{attribute 'OPC.UA.DA' := '1'}
FUNCTION_BLOCK ArduinoLight EXTENDS LightBase
VAR_INPUT
END_VAR
VAR_OUTPUT
END_VAR
VAR
	{attribute 'OPC.UA.DA' := '0'}
	_config : ArduinoLightConfig;	
	{attribute 'OPC.UA.DA' := '0'}
	_coeAccess : CoeAccess;	
	{attribute 'OPC.UA.DA' := '0'}
	_initConfigSerialCom : BOOL;	
	{attribute 'OPC.UA.DA' := '0'}
	_suffix : STRING := Const.CR_LF;
	{attribute 'OPC.UA.DA' := '0'}
	_serialCom  : SerialCom(Prefix :='', Suffix := _suffix);
	{attribute 'OPC.UA.DA' := '0'}
	_refSerialCom : REFERENCE TO SerialCom(Prefix :='', Suffix := _suffix) := _serialCom;		 
	{attribute 'OPC.UA.DA' := '0'}
	_isReceived : BOOL;
	
	{attribute 'OPC.UA.DA' := '0'}
	_deliverMessages : INT;
		
	StatusMsg : STRING(255);
	SwitchOnMsg : STRING(255);
	PowerMsg : STRING(255);
	IntensityMsg : STRING(255);	
	TemperatureMsg : STRING(255);
	LightSourcesMsg : STRING(255);
	TimeLightSourceMsg  : STRING(255);
	CustomMsg : STRING(255);
		
	{region 'Commands'}
	
	{attribute 'OPC.UA.DA' := '0'}
	_setSwitchOnCmd : BOOL;
	{attribute 'OPC.UA.DA' := '0'}
	_getSwitchOnCmd : BOOL;
	{attribute 'OPC.UA.DA' := '0'}
	_setPowerCmd : BOOL;
	{attribute 'OPC.UA.DA' := '0'}
	_getPowerCmd : BOOL;
	{attribute 'OPC.UA.DA' := '0'}
	_setIntensityCmd : BOOL;
	{attribute 'OPC.UA.DA' := '0'}
	_getIntensityCmd : BOOL;
	{attribute 'OPC.UA.DA' := '0'}
	_getTimeLightSourceCmd : BOOL;
	{attribute 'OPC.UA.DA' := '0'}
	_getLightSourcesCmd : BOOL;
	{attribute 'OPC.UA.DA' := '0'}
	_customCmd : BOOL;
	{attribute 'OPC.UA.DA' := '0'}			  		   
	_raisePropertiesCmd : BOOL;
	
	{attribute 'OPC.UA.DA' := '0'}
	_lightId : STRING; 
	{attribute 'OPC.UA.DA' := '0'}
	_switchOn : BOOL;
	{attribute 'OPC.UA.DA' := '0'}
	_setPower : LREAL;
	{attribute 'OPC.UA.DA' := '0'}
	_setIntensity : LREAL;
	{attribute 'OPC.UA.DA' := '0'}
	_cmd : STRING;	
		 
	{endregion}			
	
	{attribute 'OPC.UA.DA' := '0'}
	_initDevice : BOOL;	
	 
	{attribute 'OPC.UA.DA' := '0'}
	_lightSources : ARRAY [0..Const.PHOTOLUM_NUMBER_LIGHT_SOURCE] OF STRING(255);  
	
	{attribute 'OPC.UA.DA' := '0'}
	_itemScheduler : INT;
	{attribute 'OPC.UA.DA' := '0'}
	_itemInitScheduler : INT;
	{attribute 'OPC.UA.DA' := '0'}
	_itemExecScheduler : INT;		
	{attribute 'OPC.UA.DA' := '0'}
	_itemRaisedProperties : INT;			
	{attribute 'OPC.UA.DA' := '0'}
	_pulseGenerator : TON;	
	{attribute 'OPC.UA.DA' := '0'}
	_initPulseGenerator : TON;	
	{attribute 'OPC.UA.DA' := '0'}	
	_execPulseGenerator : TON;	
	
	{attribute 'OPC.UA.DA' := '0'}
	message : STRING;
	{attribute 'OPC.UA.DA' := '0'}
	lastMessage : STRING;	
	{attribute 'OPC.UA.DA' := '0'}
	sSubStr4 : STRING(4) := '';			
	{attribute 'OPC.UA.DA' := '0'}
	stringLength : INT;
	{attribute 'OPC.UA.DA' := '0'}
	_numberOfElements : DINT;
	{attribute 'OPC.UA.DA' := '0'}
	_indexNumberOfElements : INT;
END_VAR

IF NOT InitConfigSerialCom THEN
	ConfigureSerialCom();
ELSIF THIS^.Status = TExecutionState.Ready THEN
	SUPER^();	

	IF _refSerialCom.ErrorReceiveId = COMERROR_NOERROR THEN
		_refSerialCom(TxBuffer:= HardwareGlobalVariables.TxBufferLight, 
		 	      	  RxBuffer:= HardwareGlobalVariables.RxBufferLight);
	END_IF				  
	
	// Init device
	InitDevice();		  				 
	
	IF StateMsg <> ANY_TO_STRING(State) THEN
		StateMsg := ANY_TO_STRING(State);
	END_IF
	
	// Deliver messages
	IF _refSerialCom.IsReceived THEN	
		lastMessage := _refSerialCom.LastReceivedString;			
		stringLength := LEN(lastMessage);
		
		IF stringLength > 2 THEN
			message := LEFT(lastMessage, stringLength - 2);
		ELSE
			message := ' ';
		END_IF; 	
			
		CASE _deliverMessages OF			
			EFeedbackMsgArduinoLight.SwitchOnMsg :
				SwitchOnMsg := message;	
			EFeedbackMsgArduinoLight.PowerMsg :
				PowerMsg := message;	
			EFeedbackMsgArduinoLight.IntensityMsg :
				IntensityMsg := message;	
			EFeedbackMsgArduinoLight.TemperatureMsg :
				TemperatureMsg := message;	
			EFeedbackMsgArduinoLight.LightSourcesMsg :
				LightSourcesMsg := message;			
				_logger.Information(_message.Reset().Append('LightSourcesMsg: ').Append(LightSourcesMsg).ToString());	
			EFeedbackMsgArduinoLight.TimeLightSourceMsg :
				TimeLightSourceMsg := message;	
			EFeedbackMsgArduinoLight.CustomMsg :
				CustomMsg := message;	
		END_CASE
		
		_deliverMessages := 0;
	END_IF								   							   	
		
	SetSwitchOn(_setSwitchOnCmd, _lightId, _switchOn); 
	GetSwitchOn(_getSwitchOnCmd, _lightId);
	SetPower(_setPowerCmd, _lightId, _setPower);
	GetPower(_getPowerCmd, _lightId);
	SetIntensity(_setIntensityCmd, _lightId, _setIntensity);
	GetIntensity(_getIntensityCmd, _lightId);
	GetTimeLightSource(_getTimeLightSourceCmd, _lightId);
	GetLightSources(_getLightSourcesCmd);
	CustomCommand(_customCmd, _cmd);
	RaisePropertiesChanged(_raisePropertiesCmd, _lightId);
	
	IF _initDevice AND NOT _setSwitchOnCmd AND NOT _getSwitchOnCmd AND NOT _setPowerCmd AND NOT _getPowerCmd AND NOT _setIntensityCmd AND NOT _getIntensityCmd
	   AND NOT _getTimeLightSourceCmd AND NOT _getLightSourcesCmd AND NOT _customCmd AND NOT _raisePropertiesCmd THEN
		MessageScheduler();
	END_IF
END_IF

METHOD ConfigureSerialCom
VAR_INPUT
END_VAR
IF _coeAccess.CoeOperation.Ready THEN
	_logger.Information(_message.Reset().Append('Start configuration com serial').ToString());
END_IF;	

_coeAccess.CoeOperation.Start();
_coeAccess(SerialCommunication := _config.SerialCommunication);
	
IF _coeAccess.CoeOperation.Done THEN
	_coeAccess.SetDone();	
	
	_Logger.Information(_message.Reset().
							Append('{').Append(TO_STRING(THIS^.Family)).Append('} : ').
							Append(' - Status : ').Append(TO_STRING(_coeAccess.Status)).ToString());	
	InitConfigSerialCom := TRUE;
END_IF
 
IF _coeAccess.CoeOperation.Error THEN	
	_coeAccess.SetError(0);
	
	_Logger.Error(_message.Reset().
							Append('{').Append(TO_STRING(THIS^.Family)).Append('} : ').
							Append(' - Status : ').Append(TO_STRING(_coeAccess.Status)).ToString());
	InitConfigSerialCom := TRUE;
END_IF

THIS^.Status := _coeAccess.Status;
State := _coeAccess.Status;
END_METHOD

{attribute 'TcRpcEnable' := '1'}
(** Custom command **)
METHOD CustomCommand
VAR_INPUT
	Execute : BOOL;
	Cmd : STRING;
END_VAR
IF Execute THEN
	_logger.Information(_message.Reset().Append(_config.Name).Append(' - Custom command : ').Append(Cmd).ToString());	
	_deliverMessages := EFeedbackMsgArduinoLight.CustomMsg;														
	_serialCom.Send(Cmd);	
	_customCmd := FALSE;
END_IF
END_METHOD

METHOD FB_init : BOOL
VAR_INPUT
	bInitRetains : BOOL; // if TRUE, the retain variables are initialized (warm start / cold start)
	bInCopyCode : BOOL;  // if TRUE, the instance afterwards gets moved into the copy code (online change)
	Config : ArduinoLightConfig;
END_VAR
IF Config.IsEnabled THEN
	_config := Config;
	
	SUPER^._lightConfig.Name := Config.Name;
	SUPER^._lightConfig.DeviceID := Config.DeviceID;
	SUPER^._lightConfig.IsEnabled := Config.IsEnabled;
	SUPER^._lightConfig.LogLevel := Config.LogLevel;
	
	SUPER^.Name := Config.Name;
	SUPER^.DeviceID := Config.DeviceID;	
	THIS^.Family := DeviceFamily.Light;
		
	_Logger.Information(_message.Reset().Append('Init ').
							Append('{').Append(TO_STRING(THIS^.Family)).Append('} - ').
							Append('{').Append(TO_STRING(Config.Name)).Append('}').ToString());																													
END_IF
END_METHOD

{attribute 'TcRpcEnable' := '1'}
METHOD GetIntensity
VAR_INPUT
	Execute : BOOL;
	LightId : STRING;
END_VAR
VAR
	cmd : STRING := '*amps ';
END_VAR
IF Execute THEN	
	_deliverMessages := EFeedbackMsgArduinoLight.IntensityMsg;
	_lightId := LightId;
	_serialCom.Send(CONCAT(cmd, TO_STRING(_lightId)));
	
	_getIntensityCmd := FALSE;
END_IF
END_METHOD

METHOD GetLightSources
VAR_INPUT
	Execute: BOOL;
END_VAR
VAR
	cmd : STRING := '*list';
END_VAR
IF Execute THEN
	_logger.Information(_message.Reset().Append(_config.Name).Append(' - GetLightSources').ToString());
	_deliverMessages := EFeedbackMsgArduinoLight.LightSourcesMsg;
	_serialCom.Send(cmd);	
	
	_getLightSourcesCmd := FALSE;
END_IF
END_METHOD

{attribute 'TcRpcEnable' := '1'}
METHOD GetPower
VAR_INPUT
	Execute : BOOL;
	LightId : STRING;
END_VAR
VAR
	cmd : STRING := '*power ';
END_VAR
IF Execute THEN	
	_deliverMessages := EFeedbackMsgArduinoLight.PowerMsg;
	_lightId := LightId;
	_serialCom.Send(CONCAT(cmd, TO_STRING(_lightId)));
	
	 _getPowerCmd := FALSE;
END_IF
END_METHOD

{attribute 'TcRpcEnable' := '1'}
METHOD GetSwitchOn
VAR_INPUT
	Execute : BOOL;
	LightId : STRING;
END_VAR
VAR
	cmd : STRING := '*swit ';
END_VAR
IF Execute THEN	
	_deliverMessages := EFeedbackMsgArduinoLight.SwitchOnMsg;
	_lightId := LightId;
	_serialCom.Send(CONCAT(cmd, TO_STRING(_lightId)));
				
	_getSwitchOnCmd := FALSE;	
END_IF
END_METHOD

METHOD GetTemperature
VAR_INPUT
	LightId : STRING;
END_VAR
VAR
	cmd : STRING := '*temp ';
END_VAR
_deliverMessages := EFeedbackMsgArduinoLight.TemperatureMsg;
_lightId := LightId;
_serialCom.Send(CONCAT(cmd, _lightId));
END_METHOD

METHOD GetTimeLightSource
VAR_INPUT
	Execute: BOOL;
	LightId : STRING;
END_VAR
VAR
	cmd : STRING := '*time ';
END_VAR
IF Execute THEN
	_lightId := LightId;
	_logger.Information(_message.Reset().Append(_config.Name).Append(' - GetTimeLightSource - ').Append(TO_STRING(_lightId)).ToString());
	_deliverMessages := EFeedbackMsgArduinoLight.TimeLightSourceMsg;
	_serialCom.Send(CONCAT(cmd, _lightId));	
	
	_getTimeLightSourceCmd := FALSE;
END_IF
END_METHOD

PROPERTY InitConfigSerialCom : BOOL
GET
InitConfigSerialCom := _initConfigSerialCom;
END_GET
SET
_initConfigSerialCom := InitConfigSerialCom;
END_SET
END_PROPERTY

METHOD InitDevice
VAR_INPUT
END_VAR
VAR
	numElements : INT := 0;
    commaPos : INT;
    tempStr : STRING; 
	Separator : STRING := ',';
END_VAR
IF NOT _initDevice THEN	
	IF _initPulseGenerator.Q THEN
		_initPulseGenerator(IN := FALSE, PT := T#10MS);
			
		CASE _itemInitScheduler OF					
			0:	_logger.Information(_message.Reset().Append(_config.Name).Append(' - Init device').ToString());
				//_getLightSourcesCmd := TRUE;
				_itemInitScheduler := 50;
			
			1:	IF LightSourcesMsg <> '' THEN				
					tempStr := LightSourcesMsg;
					WHILE (LEN(tempStr) > 0) DO
						commaPos := FIND(tempStr, Separator);
						IF commaPos > 0 THEN
							_lightSources[numElements] := LEFT(tempStr, commaPos - 1);						
							tempStr := RIGHT(tempStr, LEN(tempStr) - commaPos);
						ELSE
							_lightSources[numElements] := tempStr;
							tempStr := ''; 
						END_IF
						_logger.Information(_message.Reset().Append(_config.Name).Append(' - ').Append(TO_STRING(numElements)).Append(': ').Append(_lightSources[numElements]).ToString());
						numElements := numElements + 1;						
					END_WHILE
														
					IF (numElements - 1) <> 0 THEN
						_numberOfElements := numElements;
						//_itemInitScheduler := 10; GVA
						_itemInitScheduler := 50;
					ELSE
						_itemInitScheduler := 40;	
					END_IF				
					
					_deliverMessages := -1;
				END_IF
			
			10: IF (_indexNumberOfElements >= 0) AND (_indexNumberOfElements < _numberOfElements) THEN
					tempStr := CONCAT(_lightSources[_indexNumberOfElements], ' 0');
					_serialCom.Send(CONCAT('*power ', tempStr));				
					_logger.Information(_message.Reset().Append(_config.Name).Append(' - ').Append(_lightSources[_indexNumberOfElements]).Append(' - Power: 0').ToString());	
					_indexNumberOfElements := _indexNumberOfElements + 1;
					
				ELSE
					_indexNumberOfElements := 0;
					_itemInitScheduler := 11;					
				END_IF	
			
			11: IF (_indexNumberOfElements >= 0) AND (_indexNumberOfElements < _numberOfElements) THEN
					tempStr := CONCAT(_lightSources[_indexNumberOfElements], ' 1');
					_serialCom.Send(CONCAT('*swit ', tempStr));
					_logger.Information(_message.Reset().Append(_config.Name).Append(' - ').Append(_lightSources[_indexNumberOfElements]).Append(' - Switch ON').ToString());
					_indexNumberOfElements := _indexNumberOfElements + 1;					
				ELSE
					_indexNumberOfElements := 0;
					_itemInitScheduler := 50;
				END_IF	

			41: _logger.Error(_message.Reset().Append(_config.Name).Append(' - numElements is empty: ').ToString());
				_itemInitScheduler := 50;	
		
			50: _initDevice := TRUE;
				_itemInitScheduler := 0;	
				_logger.Information(_message.Reset().Append(_config.Name).Append(' - Init device done').ToString());	
		END_CASE
	ELSE
		_initPulseGenerator(IN := TRUE, PT := T#100MS);		
	END_IF	
END_IF
END_METHOD

METHOD MessageScheduler
VAR_INPUT
END_VAR
IF _pulseGenerator.Q THEN
	_pulseGenerator(IN := FALSE, PT := T#10MS);
		
	CASE _itemScheduler OF					
		0:	IF _lightID <> '' THEN
				//GetTemperature(_lightID);
			END_IF
				
			_itemScheduler := 0;		
	END_CASE
ELSE
	_pulseGenerator(IN := TRUE, PT := T#100MS);		
END_IF


IF _pulseIsAliveGenerator.Q THEN
	_pulseIsAliveGenerator(IN := FALSE, PT := T#10MS);
		
	IsAlive();	
ELSE
	_pulseIsAliveGenerator(IN := TRUE, PT := T#1000MS);		
END_IF
END_METHOD

{attribute 'TcRpcEnable' := '1'}
METHOD RaisePropertiesChanged
VAR_INPUT
	Execute : BOOL;
	LightId : STRING;
END_VAR
VAR
	numElements : INT := 0;
    commaPos : INT;
    tempStr : STRING; 
	Separator : STRING := ',';
END_VAR
IF Execute THEN
	_raisePropertiesCmd := TRUE;
	_lightId := LightId;
	
	IF _pulseGenerator.Q THEN
		_pulseGenerator(IN := FALSE, PT := T#10MS);	

		CASE _itemRaisedProperties OF
			0:  SwitchOnMsg := ' ';
				PowerMsg := ' ';		
				IntensityMsg := ' ';
				LightSourcesMsg := ' ';		
				TimeLightSourceMsg := ' ';		
				_itemRaisedProperties := 1;					

			1:  IF _lightId <> '' THEN
					_itemRaisedProperties := 10;	
				ELSE
					_itemRaisedProperties := 40;	
				END_IF
				
			10: _getSwitchOnCmd := TRUE;													
				_itemRaisedProperties := 11;
				
			11: IF SwitchOnMsg <> ' ' THEN
					_itemRaisedProperties := 12;
				END_IF	
				
			12: _getPowerCmd := TRUE;													
				_itemRaisedProperties := 13;
				
			13: IF PowerMsg <> ' ' THEN
					_itemRaisedProperties := 14;
				END_IF
				
			14: _getIntensityCmd := TRUE;													
				_itemRaisedProperties := 15;
				
			15: IF IntensityMsg <> ' ' THEN
					_itemRaisedProperties := 16;
				END_IF
			
			16: _getTimeLightSourceCmd := TRUE;													
				_itemRaisedProperties := 17;
				
			17: IF TimeLightSourceMsg <> ' ' THEN
					_itemRaisedProperties := 50;
				END_IF
			
			40: _logger.Error(_message.Reset().Append(_config.Name).Append(' - RaisePropertiesChanged - LightId is empty').ToString());
				_itemRaisedProperties := 50;
			
			50:  _logger.Information(_message.Reset().Append(_config.Name).Append(' - RaisePropertiesChanged').ToString());
				_raisePropertiesCmd := FALSE;				
				_itemRaisedProperties := 0;
			
		END_CASE
	ELSE
		_pulseGenerator(IN := TRUE, PT := T#50MS);	
	END_IF
END_IF
END_METHOD

{attribute 'TcRpcEnable' := '1'}
METHOD SetIntensity
VAR_INPUT
	Execute : BOOL;
	LightId : STRING;
	Intensity : LREAL;
END_VAR
VAR
	cmd : STRING := '*amps ';
	tmpConcatLightIdIntensity : STRING;
END_VAR
IF Execute THEN	
	_setIntensityCmd := TRUE;
	_lightId := LightId;
	_setIntensity := Intensity; 
	
	IF _execPulseGenerator.Q THEN
		_execPulseGenerator(IN := FALSE, PT := T#10MS);
			
		CASE _itemExecScheduler OF
			0:  IF _lightId <> '' THEN
					_itemExecScheduler := 10;	
				ELSE
					_itemExecScheduler := 40;	
				END_IF
				
				_deliverMessages := -1;

			10: _lightId := LightId;
				tmpConcatLightIdIntensity := CONCAT(CONCAT(_lightId, ' '), TO_STRING(Intensity));

				_logger.Information(_message.Reset().Append(_config.Name).Append(' - ').Append(_lightId).Append(' - SetIntensity : ').Append(TO_STRING(_lightId)).Append(' - ').Append(TO_STRING(Intensity)).ToString());
				_serialCom.Send(CONCAT(cmd, TO_STRING(tmpConcatLightIdIntensity)));
				_itemExecScheduler := 11;
			
			11:  _getIntensityCmd := TRUE;
				_itemExecScheduler := 50;
			
			40: _logger.Error(_message.Reset().Append(_config.Name).Append(' - SetIntensity - LightId is empty').ToString());
				_itemExecScheduler := 50;
		
			50:  _setIntensityCmd := FALSE;	
				_itemExecScheduler := 0;		
								
		END_CASE
	ELSE
		_execPulseGenerator(IN := TRUE, PT := T#100MS);	
	END_IF
END_IF
END_METHOD

{attribute 'TcRpcEnable' := '1'}
METHOD SetPower
VAR_INPUT
	Execute : BOOL;
	LightId : STRING;
	Power : LREAL;
END_VAR
VAR
	cmd : STRING := '*power ';
	tmpConcatLightIdPower : STRING;
END_VAR
IF Execute THEN	
	_setPowerCmd := TRUE;	
	_lightId := LightId;
	_setPower := Power;	
	
	IF _execPulseGenerator.Q THEN
		_execPulseGenerator(IN := FALSE, PT := T#10MS);
			
		CASE _itemExecScheduler OF
			0:  IF _lightId <> '' THEN
					_itemExecScheduler := 10;	
				ELSE
					_itemExecScheduler := 40;	
				END_IF
				
				_deliverMessages := -1;

			10: _lightId := LightId;
				tmpConcatLightIdPower := CONCAT(CONCAT(_lightId, ' '), TO_STRING(Power));

				_logger.Information(_message.Reset().Append(_config.Name).Append(' - ').Append(_lightId).Append(' - SetPower : ').Append(TO_STRING(Power)).ToString());
				_serialCom.Send(CONCAT(cmd, TO_STRING(tmpConcatLightIdPower)));
				_itemExecScheduler := 11;
			
			11:  _getPowerCmd := TRUE;
				_itemExecScheduler := 50;
			
			40: _logger.Error(_message.Reset().Append(_config.Name).Append(' - SetPower - LightId is empty').ToString());
				_itemExecScheduler := 50;
	
			50:  _setPowerCmd := FALSE;	
				_itemExecScheduler := 0;		
								
		END_CASE
	ELSE
		_execPulseGenerator(IN := TRUE, PT := T#100MS);	
	END_IF
END_IF
END_METHOD

{attribute 'TcRpcEnable' := '1'}
METHOD SetSwitchOn
VAR_INPUT
	Execute : BOOL;	
	LightId : STRING;
	SwitchOn : BOOL;
END_VAR
VAR
	cmd : STRING := '*swit ';
	tmpConcatLightIdSwitchOn : STRING;
	tmp : STRING;
	switchOnValue : STRING;
END_VAR
IF Execute THEN	
	_setSwitchOnCmd := TRUE;	
	_switchOn := SwitchOn; 
	_lightId := LightId;
	
	IF _execPulseGenerator.Q THEN
		_execPulseGenerator(IN := FALSE, PT := T#10MS);
			
		CASE _itemExecScheduler OF
			0:  IF _lightId <> '' THEN
					_itemExecScheduler := 10;	
				ELSE
					_itemExecScheduler := 40;	
				END_IF
				
				_deliverMessages := -1;

			10:	_lightId := LightId;				
			
				IF _switchOn THEN
					switchOnValue := '1';
				ELSE
					switchOnValue := '0';
				END_IF
				tmpConcatLightIdSwitchOn := CONCAT(CONCAT(_lightId, ' '), TO_STRING(switchOnValue));
				
				_logger.Information(_message.Reset().Append(_config.Name).Append(' - ').Append(_lightId).Append(' - SwitchOn : ').Append(TO_STRING(switchOnValue)).ToString());
				tmp := CONCAT(cmd, TO_STRING(tmpConcatLightIdSwitchOn));
				_serialCom.Send(tmp);
				_itemExecScheduler := 11;
			
			11:  _getSwitchOnCmd := TRUE;
				_itemExecScheduler := 50;
				
			40: _logger.Error(_message.Reset().Append(_config.Name).Append(' - SwitchOn - LightId is empty').ToString());
				_itemExecScheduler := 50;
				
			50:  _setSwitchOnCmd := FALSE;	
				_switchOn := FALSE;
				_itemExecScheduler := 0;		
								
		END_CASE
	ELSE
		_execPulseGenerator(IN := TRUE, PT := T#200MS);	
	END_IF
END_IF
END_METHOD

END_FUNCTION_BLOCK

(* stored: Version 1.1.0.1, ProductVersion 3.1.4024.12
   POU ArduinoLight: Id {41131ff7-9fb0-4ea7-b4b5-61dc0d90618d}, SpecialFunc None
   Folder Commands: Id {175611c0-1c97-4f96-9d9e-23c8a9dc165b}
   Method ConfigureSerialCom: Id {a6d1b958-3d6c-4736-904e-410ef01c391a}
   Method CustomCommand: Id {a874ab95-6445-4e1e-9fcb-6a865b85d7bd}
   Method FB_init: Id {607a0c2f-c498-421f-a197-39698ae4d3aa}
   Method GetIntensity: Id {895d119c-2d50-4d8d-9a46-7c78b10f3326}
   Method GetLightSources: Id {be18b0b2-340b-437e-ace2-b68eeaecd6bf}
   Method GetPower: Id {de1d776a-f167-4907-8088-a5a90ac0d59d}
   Method GetSwitchOn: Id {47b2e75a-687b-4be0-bfbb-d974608c9f4e}
   Method GetTemperature: Id {e1145ce5-e7b6-4fee-862e-5735b5e0188d}
   Method GetTimeLightSource: Id {a07dd3a1-aa20-47ef-91f8-276328c4a28c}
   Property InitConfigSerialCom: Id {c9ed0883-576d-4619-9db9-425e052b5c8e}
   Get Get: Id {bd3383a6-9bec-41f8-a2ab-436b3ebf1e55}
   Set Set: Id {279f8fb8-20b9-4936-a59d-19adfb60b9e7}
   Method InitDevice: Id {f5b8243b-1b57-4903-9f91-10352f04fca5}
   Method MessageScheduler: Id {ef7c515f-263a-4832-88bd-bd96336c6a50}
   Method RaisePropertiesChanged: Id {8027495e-3aad-4491-8af4-b8f2b2267389}
   Method SetIntensity: Id {8796987f-ba95-4a7b-ad40-343105ec6729}
   Method SetPower: Id {ad6db274-b958-4481-b7b4-94e8f4463dac}
   Method SetSwitchOn: Id {6bea85ae-da1b-4487-81c2-75ee0d05e520} *)
